// Brief: Setup Arm Init
FUNCTION_BLOCK PUBLIC FB_SetupCtrlMasterSlave EXTENDS FB_SetupArmCtrlBase
VAR_INPUT
END_VAR
VAR_OUTPUT
END_VAR
VAR
	m_initState :INT :=0;
END_VAR

END_FUNCTION_BLOCK

(* stored: Version 1.1.0.1, ProductVersion 3.1.4024.11
   POU FB_SetupCtrlMasterSlave: Id {5c90b003-cbb0-4300-8cbb-c2de7aca85f9}, SpecialFunc None *)
